// TIA Portal V20 export
DATA_BLOCK "DB_DecodChannels"   // DB405
{ DB_Accessible_From_OPC_UA := 'FALSE' }
AUTHOR : BAJ
// stored: AutoNumber false, DBAccessibleFromOPCUA false, DBAccessibleFromWebserver false, InstanceOfName FB_DecodChannels, InstanceOfType FB
"FB_DecodChannels"
   // VAR
   //    sChan1IsDisplayed : Bool;
   //    sChan2IsDisplayed : Bool;
   //    sChan3IsDisplayed : Bool;
   //    sChan4IsDisplayed : Bool;
   // END_VAR
BEGIN
END_DATA_BLOCK
